(* IEC 61131-3 sources: RL_MAR/experiments/comparison/autoplc/results/qwen3.5-9b_20260511_180311/med_30, 1 file *)

(* ---- med_30_1.st ---- *)
FUNCTION_BLOCK MuseumClimateControl
VAR_INPUT
    HumiditySensor : REAL;
    TemperatureSensor : REAL;
    LightSensor : BOOL;
END_VAR
VAR_OUTPUT
    HVACSystem : BOOL;
    Humidifier : BOOL;
    Dehumidifier : BOOL;
    LightControl : BOOL;
END_VAR
VAR
    TargetHumidity : REAL := 50.0;
    TargetTemperature : REAL := 20.0;
    LightThreshold : BOOL := TRUE;
END_VAR

IF HumiditySensor < TargetHumidity THEN
    Humidifier := TRUE;
    Dehumidifier := FALSE;
ELSIF HumiditySensor > TargetHumidity THEN
    Dehumidifier := TRUE;
    Humidifier := FALSE;
ELSE
    Humidifier := FALSE;
    Dehumidifier := FALSE;
END_IF;

IF TemperatureSensor <> TargetTemperature THEN
    HVACSystem := TRUE;
ELSE
    HVACSystem := FALSE;
END_IF;

IF LightSensor = TRUE AND LightThreshold = TRUE THEN
    LightControl := FALSE;
ELSE
    LightControl := TRUE;
END_IF;

END_FUNCTION_BLOCK
